FUNCTION alg_a_handlingready : BOOL
VAR_INPUT
	state: STATE;
END_VAR

alg_a_handlingready := FALSE;

END_FUNCTION

(* stored: Version 1.1.0.1, ProductVersion 3.1.4022.18
   POU alg_a_handlingready: Id {e433313a-1b96-45e8-ac4d-471f9ba068c4}, SpecialFunc None *)
